// TIA Portal V18 export
TYPE "Bound_ShW"
// stored: IsFailsafeCompliant false
   STRUCT
      Trigger : Bool;
      MainID : String[48];
      CarrierID : Int;
      Completed : Bool;
      Result : Int;
   END_STRUCT;
END_TYPE
